FUNCTION_BLOCK overcurrent (* Basic Function Block Type *)
  (* Standard: 61499-2 *)
  (* Version 0.0, 21/03/2016, Chen-Wei, nxtControl GmbH, Template *)
  PACKAGE Main;
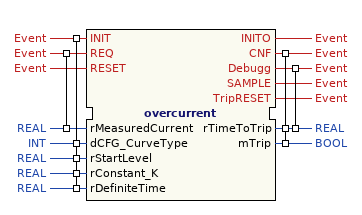
  EVENT_INPUT
    INIT WITH dCFG_CurveType, rStartLevel, rConstant_K, rDefiniteTime; (* Initialization Request *)
    REQ WITH rMeasuredCurrent; (* Normal Execution Request *)
    RESET;
  END_EVENT
  EVENT_OUTPUT
    INITO; (* Initialization Confirm *)
    CNF WITH rTimeToTrip, mTrip; (* Execution Confirmation *)
    Debugg WITH rTimeToTrip;
    SAMPLE;
    TripRESET;
  END_EVENT
  VAR_INPUT
    rMeasuredCurrent : REAL; (* Input event qualifier *)
    dCFG_CurveType : INT;
    rStartLevel : REAL;
    rConstant_K : REAL;
    rDefiniteTime : REAL;
  END_VAR
  VAR_OUTPUT
    rTimeToTrip : REAL;
    mTrip : BOOL;
  END_VAR
  VAR
    mStart : BOOL;
  END_VAR
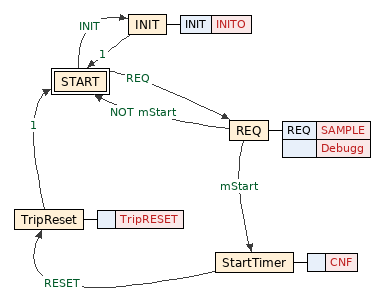
  EC_STATES
    START; (* Initial State *)
    INIT : INIT -> INITO; (* Initialization *)
    REQ : REQ -> SAMPLE, -> Debugg; (* Normal execution *)
    StartTimer : -> CNF;
    TripReset : -> TripRESET;
  END_STATES
  EC_TRANSITIONS
    START TO INIT := INIT;
    INIT TO START := 1;
    START TO REQ := REQ;
    StartTimer TO TripReset := RESET;
    REQ TO START := NOT mStart;
    REQ TO StartTimer := mStart;
    TripReset TO START := 1;
  END_TRANSITIONS
  ALGORITHM INIT IN ST: (* Initialization algorithm *)
INIT := 0;
mStart := FALSE;
;
  END_ALGORITHM
  ALGORITHM REQ IN ST: (* Normally executed algorithm Version:      1.04 2016-03-21 First Version Curvtype: (dCFG_CurveType) 0 : Definite time 1: IEC Normal Inverse 2: IEC Very Inverse 3: IEC Extremely Inverse 4: RI Curve *)
VAR
	ans1:REAL;
	ans2:REAL;
	ans3:REAL;
	veryLargeNumber:REAL:= 9999999;
END_VAR;

REQ := 0;

IF (rMeasuredCurrent >= rStartLevel) THEN
	(* The current is over start level (pickup) *)
	mStart:=TRUE;
ELSIF (rMeasuredCurrent < ( rStartLevel * 0.95 )) THEN
	(* Under start level *)
	mStart:=FALSE;
	rTimeToTrip:=0.0;
	(* IF tmrTripPulse.Q THEN
		mTrip:=FALSE;
	END_IF; *)
END_IF;

IF mStart THEN
		(* Calculate time to trip *)
	CASE dCFG_CurveType OF
		1: (* IEC Normal Inverse *)

		IF (rStartLevel = 0.0) THEN
			ans1 := EXPT(veryLargeNumber, 0.02);
		ELSE
			ans1 := EXPT((rMeasuredCurrent/rStartLevel) , 0.02);
		END_IF;

		IF ((ans1 - 1.0) = 0.0) THEN
		  ans2 := veryLargeNumber;
		ELSE
		  ans2 := 0.14/(ans1 - 1.0);
		END_IF;
		rTimeToTrip := rConstant_K*ans2;
		mTrip := TRUE;

		2: (* IEC Very Inverse *)

		IF (rStartLevel = 0.0) THEN
			ans1 := veryLargeNumber - 1.0;
		ELSE
			ans1 := (rMeasuredCurrent/rStartLevel) - 1.0;
		END_IF;

		IF (ans1 = 0.0) THEN
		  ans2 := veryLargeNumber;
		ELSE
		  ans2 := 13.5/ans1;
		END_IF;
		rTimeToTrip := rConstant_K*ans2;
		mTrip := TRUE;

		3: (* IEC Extremely Inverse *)

		IF (rStartLevel = 0.0) THEN
			ans1 := EXPT(veryLargeNumber, 2.0);
		ELSE
			ans1 := EXPT((rMeasuredCurrent/rStartLevel) , 2.0);
		END_IF;

		IF ((ans1 - 1.0) = 0.0) THEN
		  ans2 := veryLargeNumber;
		ELSE
		  ans2 := 80.0/(ans1 - 1.0);
		END_IF;
		rTimeToTrip := rConstant_K*ans2;
		mTrip := TRUE;

		4: (* RI Curve *)

		IF (rStartLevel = 0.0) THEN
			ans1 := veryLargeNumber;
		ELSE
			ans1 := rMeasuredCurrent/rStartLevel;
		END_IF;

		IF (ans1 = 0.0) THEN
		  ans2 := veryLargeNumber;
		ELSE
		  ans2 := 0.339-(0.236/ans1);
		END_IF;

		IF (ans2 = 0.0) THEN
			ans3 := veryLargeNumber;
		ELSE
			ans3 := (1.0/ans2);
		END_IF;

		rTimeToTrip := rConstant_K*ans3;
		mTrip := TRUE;

		ELSE
			(* Definite Time *)
			rTimeToTrip := rDefiniteTime;
			mTrip := TRUE;
	END_CASE;

END_IF;


;
  END_ALGORITHM
  ALGORITHM RESET IN ST:
mStart := FALSE;

;
  END_ALGORITHM
  ALGORITHM CalculateTime IN ST:
;
  END_ALGORITHM
END_FUNCTION_BLOCK
